FUNCTION_BLOCK FB_TaskMoveB_tilt EXTENDS FB_AbstructFuture
VAR_OUTPUT
END_VAR
VAR
	_v				: MC_LREAL;
	_a				: MC_LREAL;
	_d				: MC_LREAL;
	_j				: MC_LREAL;
	_dynamics		: DynamicConstraint_PathXY;
	_position 		: LREAL;
	_error_id		: UDINT;
	_fbMover		: POINTER TO MC_PlanarMover;
	_cmdFB			: MC_PlanarFeedback;
	_prohibit 		: BOOL;
	_abort_executor : FB_Executor;
	_state_num 			:UINT;
	_abort_state	:UINT;
END_VAR

{warning 'add method implementation '}
METHOD abort : BOOL
VAR_INST
	home_a :BOOL;
	home_b :BOOL;
END_VAR
_cmdFB.Update();
_state_num :=0;
CASE _abort_state OF
	0:
		IF _cmdFB.Active THEN
			_dynamics.SetValuesVADJ(2000,20000,200000,200000);
			home_a := FALSE;
			home_b := FALSE;
			//停止
			_fbMover^.Halt(_cmdFB,_dynamics);
			_abort_state := 1;
		ELSE
			abort := TRUE;
		END_IF
	1:
		IF _cmdFB.Done THEN
			IF _cmdFB.Error THEN
				abort := TRUE;
				_abort_state := 0;
				_error_id := _cmdFB.ErrorId;
			ELSE
				IF NOT home_a THEN
					_abort_state := 2;
				ELSIF NOT home_b THEN
					_abort_state := 3;
				ELSE
					abort := TRUE;
					_error_id := 0;
				END_IF
			END_IF
		END_IF
	2:
		_fbMover^.MoveA(_cmdFB,0,_dynamics);
		home_a := TRUE;
		_abort_state := 1;
	3:
		_fbMover^.MoveB(_cmdFB,0,_dynamics);
		home_b := TRUE;
		_abort_state := 1;
END_CASE
END_METHOD

{warning 'add method implementation '}
METHOD execute : BOOL
_cmdFB.Update();
_abort_state := 0;
CASE _state_num OF
	0:
		//直線運動
		IF NOT _cmdFB.Active AND NOT _cmdFB.Busy THEN
			_fbMover^.MoveB(_cmdFB,_position,_dynamics);
			_state_num := 1;
		END_IF
	1:
		//直線運動の完了フラグ待ち
		IF _cmdFB.Done THEN
			execute := TRUE;
			_error_id := 0;
		END_IF
		IF _cmdFB.Error THEN
			execute := TRUE;
			_error_id := _cmdFB.ErrorId;
		END_IF
END_CASE
END_METHOD

METHOD FB_init : BOOL
VAR_INPUT
	bInitRetains : BOOL; // if TRUE, the retain variables are initialized (warm start / cold start)
	bInCopyCode : BOOL;  // if TRUE, the instance afterwards gets moved into the copy code (online change)
	fbMover : REFERENCE TO MC_PlanarMover;
END_VAR
_fbMover := ADR(fbMover);
END_METHOD

{warning 'add method implementation '}
METHOD init : BOOL
IF _prohibit THEN
	_error_id := 16#80000000;
	init := TRUE;
ELSIF _v = 0 OR _a = 0 OR _d = 0 THEN
	_error_id := 1;
	init := TRUE;
ELSE
	_dynamics.SetValuesVADJ(_v, _a, _d, _j);
	_abort_executor.init();
	_error_id := 0;
	_state_num := 0;
	_abort_state := 0;
	init := TRUE;
END_IF
END_METHOD

{warning 'add property implementation'}
PROPERTY nErrorID : UDINT
GET
nErrorID := _error_id;
END_GET
END_PROPERTY

{warning 'add method implementation '}
METHOD quit : BOOL
init();
quit := TRUE;
END_METHOD

METHOD set_dynamics : BOOL
VAR_INPUT
	v: MC_LREAL;
	a: MC_LREAL;
	d: MC_LREAL;
	j: MC_LREAL;
END_VAR
_v := v;
_a := a;
_d := d;
_j := j;
set_dynamics := TRUE;
END_METHOD

METHOD set_target_position : BOOL
VAR_INPUT
	z: LREAL;
END_VAR
_position := z;

set_target_position := TRUE;
END_METHOD

END_FUNCTION_BLOCK

(* stored: Version 1.1.0.1, ProductVersion 3.1.4024.12
   POU FB_TaskMoveB_tilt: Id {0915bf68-8cd3-47f3-a868-5bca07ff999e}, SpecialFunc None
   Method abort: Id {9254f68e-e982-4783-b590-a93424860c2b}
   Method execute: Id {e7c05af9-16b9-43c4-b4ce-a49ab41c74df}
   Method FB_init: Id {a6f9218a-d462-4b39-b391-bcc06be0f17e}
   Method init: Id {0cb235b0-0cb7-47e3-9412-6ddc30f77f28}
   Property nErrorID: Id {23550152-5cf6-430c-9469-fa6b564a2c2d}
   Get Get: Id {b3113753-3c2a-4b64-9aa8-ac067a373276}
   Method quit: Id {cd971d0f-5369-431e-b1d8-48334864eed7}
   Method set_dynamics: Id {98f29237-3e72-49c7-9d44-0b205fe23fe8}
   Method set_target_position: Id {b43d0496-bd78-4589-b117-01ab25d1632f} *)
